PROGRAM Alarmes
VAR
	T1Compressor: TON;
	T2PortaAberta: TON;
	SinalIntermitente: PiscaPisca;
END_VAR

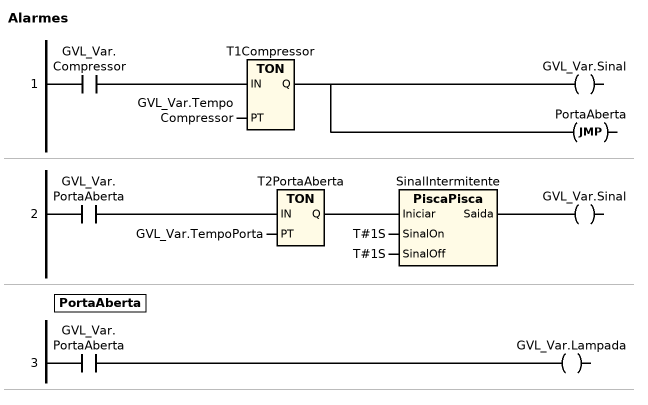
// NETWORK 1
T1Compressor(IN := GVL_Var.Compressor, PT := GVL_Var.TempoCompressor); // TON
GVL_Var.Sinal := T1Compressor.Q;
IF T1Compressor.Q THEN JMP PortaAberta; END_IF

// NETWORK 2
T2PortaAberta(IN := GVL_Var.PortaAberta, PT := GVL_Var.TempoPorta); // TON
SinalIntermitente(Iniciar := T2PortaAberta.Q, SinalOn := T#1S, SinalOff := T#1S); // PiscaPisca
GVL_Var.Sinal := SinalIntermitente.Saida;

// NETWORK 3
PortaAberta:
GVL_Var.Lampada := GVL_Var.PortaAberta;

END_PROGRAM

(* stored: Version 1.1.0.1
   POU Alarmes: Id {8746115f-edbb-4c9d-a33d-27377980ac12}, SpecialFunc None *)
